FUNCTION_BLOCK SDODatenMotor2
VAR_INPUT
END_VAR
VAR_OUTPUT
	
	Motor2Spannung: UINT;
	Motor2Strom: INT;
	Motor2Strombegrenzung: UINT;
	Motor2Regelfehler: INT;
	Motor2Geschwindigkeit: INT;
	Motor2Overloadtime: UINT;
	Motor2Overtemperature: BOOL;
	Motor2Torqueoverload: BOOL;
	Motor2Shortcirciut: BOOL;
	
END_VAR
VAR
	Motorspannung: FB_EcCoESdoRead;	
	Motorstrom: FB_EcCoESdoRead;
	Strombegrenzung: FB_EcCoESdoRead;
	Regelfehler: FB_EcCoESdoRead;
	Geschwindigkeit: FB_EcCoESdoRead;
	Overload: FB_EcCoESdoRead;
	Short_Circuit: FB_EcCoESdoRead;
	Torque_Overload: FB_EcCoESdoRead;
	Over_Temperature: FB_EcCoESdoRead;

	trigger: BOOL;
	TON_0: TON;
	TON_1: TON;
	ms: TIME;

END_VAR

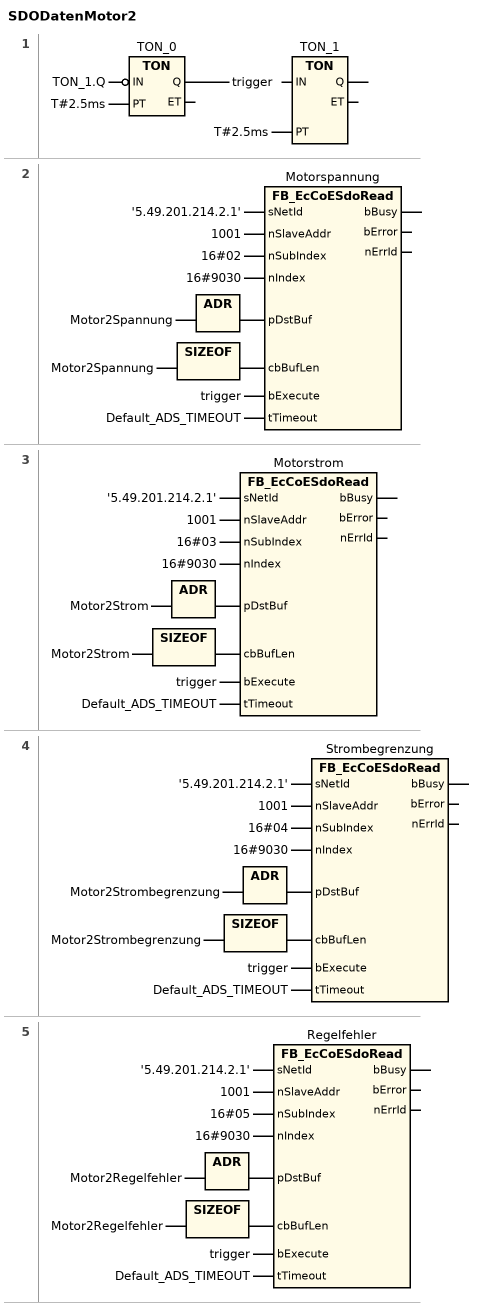
// NETWORK 1
TON_0(IN := NOT TON_1.Q, PT := T#2.5ms); // TON
trigger := TON_0.Q;
TON_1(IN := TON_0.Q, PT := T#2.5ms); // TON

// NETWORK 2
Motorspannung(
    sNetId := '5.49.201.214.2.1',
    nSlaveAddr := 1001,
    nSubIndex := 16#02,
    nIndex := 16#9030,
    pDstBuf := ADR(Motor2Spannung),
    cbBufLen := SIZEOF(Motor2Spannung),
    bExecute := trigger,
    tTimeout := Default_ADS_TIMEOUT); // FB_EcCoESdoRead

// NETWORK 3
Motorstrom(
    sNetId := '5.49.201.214.2.1',
    nSlaveAddr := 1001,
    nSubIndex := 16#03,
    nIndex := 16#9030,
    pDstBuf := ADR(Motor2Strom),
    cbBufLen := SIZEOF(Motor2Strom),
    bExecute := trigger,
    tTimeout := Default_ADS_TIMEOUT); // FB_EcCoESdoRead

// NETWORK 4
Strombegrenzung(
    sNetId := '5.49.201.214.2.1',
    nSlaveAddr := 1001,
    nSubIndex := 16#04,
    nIndex := 16#9030,
    pDstBuf := ADR(Motor2Strombegrenzung),
    cbBufLen := SIZEOF(Motor2Strombegrenzung),
    bExecute := trigger,
    tTimeout := Default_ADS_TIMEOUT); // FB_EcCoESdoRead

// NETWORK 5
Regelfehler(
    sNetId := '5.49.201.214.2.1',
    nSlaveAddr := 1001,
    nSubIndex := 16#05,
    nIndex := 16#9030,
    pDstBuf := ADR(Motor2Regelfehler),
    cbBufLen := SIZEOF(Motor2Regelfehler),
    bExecute := trigger,
    tTimeout := Default_ADS_TIMEOUT); // FB_EcCoESdoRead

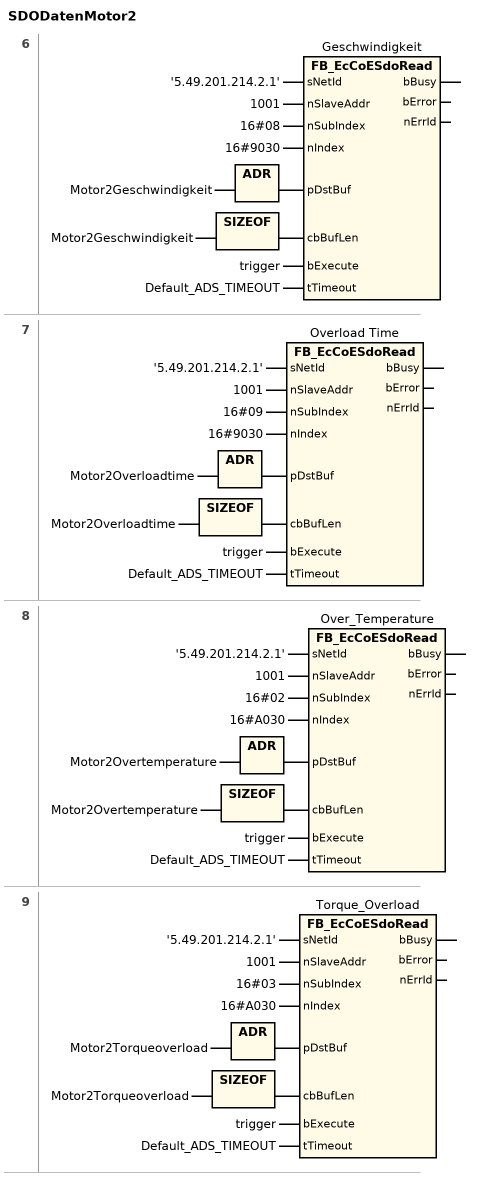
// NETWORK 6
Geschwindigkeit(
    sNetId := '5.49.201.214.2.1',
    nSlaveAddr := 1001,
    nSubIndex := 16#08,
    nIndex := 16#9030,
    pDstBuf := ADR(Motor2Geschwindigkeit),
    cbBufLen := SIZEOF(Motor2Geschwindigkeit),
    bExecute := trigger,
    tTimeout := Default_ADS_TIMEOUT); // FB_EcCoESdoRead

// NETWORK 7
Overload Time(
    sNetId := '5.49.201.214.2.1',
    nSlaveAddr := 1001,
    nSubIndex := 16#09,
    nIndex := 16#9030,
    pDstBuf := ADR(Motor2Overloadtime),
    cbBufLen := SIZEOF(Motor2Overloadtime),
    bExecute := trigger,
    tTimeout := Default_ADS_TIMEOUT); // FB_EcCoESdoRead

// NETWORK 8
Over_Temperature(
    sNetId := '5.49.201.214.2.1',
    nSlaveAddr := 1001,
    nSubIndex := 16#02,
    nIndex := 16#A030,
    pDstBuf := ADR(Motor2Overtemperature),
    cbBufLen := SIZEOF(Motor2Overtemperature),
    bExecute := trigger,
    tTimeout := Default_ADS_TIMEOUT); // FB_EcCoESdoRead

// NETWORK 9
Torque_Overload(
    sNetId := '5.49.201.214.2.1',
    nSlaveAddr := 1001,
    nSubIndex := 16#03,
    nIndex := 16#A030,
    pDstBuf := ADR(Motor2Torqueoverload),
    cbBufLen := SIZEOF(Motor2Torqueoverload),
    bExecute := trigger,
    tTimeout := Default_ADS_TIMEOUT); // FB_EcCoESdoRead

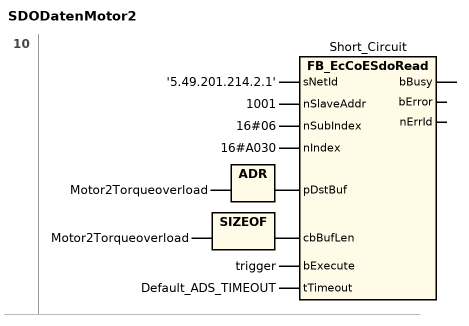
// NETWORK 10
Short_Circuit(
    sNetId := '5.49.201.214.2.1',
    nSlaveAddr := 1001,
    nSubIndex := 16#06,
    nIndex := 16#A030,
    pDstBuf := ADR(Motor2Torqueoverload),
    cbBufLen := SIZEOF(Motor2Torqueoverload),
    bExecute := trigger,
    tTimeout := Default_ADS_TIMEOUT); // FB_EcCoESdoRead

END_FUNCTION_BLOCK

(* stored: Version 1.1.0.1, ProductVersion 3.1.4020.12
   POU SDODatenMotor2: Id {fc3f6e21-44fa-4032-ac2a-99de5ee82a27}, SpecialFunc None *)
